{attribute 'linkalways'} 
{attribute 'no_explicit_call' := 'This FB is a CLASS and must be accessed using methods or properties'}
{attribute 'enable_dynamic_creation'}
FUNCTION_BLOCK StopCommand_1 EXTENDS Mc2AsyncCommand
VAR
	fb : Tc2_Mc2.Mc_Stop;
END_VAR

{attribute 'monitoring' := 'call'}
PROPERTY PUBLIC Active : BOOL
GET // PUBLIC
Active := fb.Active;
END_GET
END_PROPERTY

METHOD PUBLIC CyclicCall
SUPER^.CyclicCall();
fb(Axis := axis_ref);
END_METHOD

(*FB_Init is always available implicitly and it is used primarily for initialization.
The return value is not evaluated. For a specific influence, you can also declare the
methods explicitly and provide additional code there with the standard initialization
code. You can evaluate the return value.*)
METHOD FB_Init : BOOL
VAR_INPUT
	(* TRUE: the retain variables are initialized (reset warm / reset cold)*)
	bInitRetains : BOOL;
	(* TRUE: the instance will be copied to the copy code afterward (online change)*)
	bInCopyCode	: BOOL;
	axis : REFERENCE TO Mc2Axis;
	deceleration : LREAL := 0;
	jerk : LREAL := 0;
END_VAR
fb.Deceleration := deceleration;
fb.Jerk := jerk;
END_METHOD

METHOD PROTECTED OnExecuting
VAR_INPUT
	state_control : AsyncCommandStateControl;
END_VAR
fb.Execute := TRUE;

IF fb.Done THEN
	state_control.Next();
	fb.Execute := FALSE;
END_IF

IF fb.CommandAborted THEN
	Abort();
	fb.Execute := FALSE;
END_IF

IF fb.Error THEN
	state_control.Error(fb.ErrorId);
	fb.Execute := FALSE;
END_IF
END_METHOD

END_FUNCTION_BLOCK

(* stored: Version 1.1.0.1, ProductVersion 3.1.4026.13
   POU StopCommand_1: Id {db71aab2-8061-4d80-866e-67eb58e8a6a8}, SpecialFunc None
   Property Active: Id {b9903db8-5b4d-4867-85a8-7fba49fdd64f}
   Get Get: Id {a20d420c-6254-42ea-8d05-823e75050ada}
   Method CyclicCall: Id {6b17f833-3ad5-4050-ad22-ac50b84313d6}
   Method FB_Init: Id {7886e2a7-162c-4ebc-b641-6db7385ef135}
   Method OnExecuting: Id {52ddd194-a2d8-4295-933c-f14ce7508771} *)
